// TIA Portal V17 export
// export: Created 2025-03-07T09:18:54.2886173Z, ExportSetting WithDefaults, DisplayName Totally Integrated Automation Portal, DisplayVersion V17 Update 8, DisplayName TIA Portal Openness, DisplayVersion V17 Update 8, DisplayName TIA Portal Version Control Interface, DisplayVersion V17, DisplayName SINAMICS Startdrive Advanced, DisplayVersion V17 SP2, DisplayName SINAMICS Startdrive G110M, G120, G120C, G120D, G120P, G115D, DisplayVersion V17 SP2, DisplayName SINAMICS Startdrive G130, G150, S120, S150, SINAMICS MV, S210, DisplayVersion V17 SP2, DisplayName STEP 7 Professional, DisplayVersion V17 Update 8, DisplayName SINUMERIK ONE STEP 7 Toolbox, DisplayVersion V17 Update 12, DisplayName SINUMERIK 840D sl STEP 7 Toolbox, DisplayVersion V17 Update 12, DisplayName STEP 7 Safety, DisplayVersion V17 Update 6, DisplayName WinCC Advanced, DisplayVersion V17 Update 8
DATA_BLOCK "DB20211_TRUMPF_LASER_UNIT_02_READY"   // DB20211
{ DB_Accessible_From_OPC_UA := 'FALSE' }
VERSION : 0.1
// stored: AutoNumber false, DBAccessibleFromOPCUA false, DBAccessibleFromWebserver true, InstanceOfName FB20200_TRUMPF_READY, InstanceOfType FB
"FB20200_TRUMPF_READY"
   // VAR_INPUT
   //    iLIMIT_MIN_POWER : Int;
   //    iLIMIT_MAX_POWER : Int;
   //    iCOMMAND_POWER : Int;
   //    iCOMMAND_PROCESSING : Int;
   //    iCOMMAND_POWER_PORTION_CORE : Int;
   //    iSTATUS_READY_LASER_READY : Bool;
   //    iLASER_IS_ON : Bool;
   //    iSYSTEM_ERROR_LASER_FAULT : Bool;
   //    iEXTERNAL_CONTROL_READY : Bool;
   //    iPROGRAM_ACTIVE : Bool;
   //    iSOURCE_ENABLED : Bool;
   //    iCOOLING_UNIT_FLOW_PRESENT : Bool;
   //    iCOOLING_UNIT_OVERTEMPERATURE : Bool;
   //    iLASER_ENABLE_POWER_SEQ : Bool;
   //    iLASER_DISABLE_POWER_SEQ : Bool;
   //    iSAFETY_GATES_CLOSED_LOCKED : Bool;
   //    iLASER_ASSIGNED : Bool;
   //    iMACHINE_ON : Bool;
   //    iMACHINE_ON_DELAYED : Bool;
   //    iLASER_READY_F_CIRCUIT_BRAKER : Bool;
   //    iLASER_WARNING_LAP_ON : Bool;
   //    iSTATION_UNIT_ANY_CYCLE_ACT : Bool;
   //    iLASER_ACT_START_GEN_CONDITION : Bool;
   //    iUNIT_NO : Byte;
   // END_VAR
   // VAR_OUTPUT
   //    oLIGHT_PATH : Byte;
   //    oPROGRAM_NUMBER : Byte;
   //    oPOWER_VALUE : DInt;
   //    oPROCESSING_VALUE : DInt;
   //    oPOWER_PORTION_CORE_VALUE : DInt;
   //    oLASER_RESET_FAULT_ERROR : Bool;
   //    oLASER_REQUEST : Bool;
   //    oEXTERNAL_CONTROL : Bool;
   //    oLASER_ON : Bool;
   //    oLASER_ARM : Bool;
   //    oSTATION_RHP_SEOC_ALARMS : Bool;
   //    oSTATION_WARNING : Bool;
   //    oREADY_TO_EMISSION : Bool;
   //    oALARM_CIRCUIT_BREAKER_ALARM : Bool;
   //    oALARM_LASER_ERROR : Bool;
   //    oALARM_WARNING_LASER : Bool;
   //    oALARM_LASER_NOT_READY : Bool;
   //    oALARM_LASER_NOT_SWITCHED_ON : Bool;
   //    oALARM_ANALOG_CONTROL_ERROR : Bool;
   //    oALARM_LASER_NOT_ASSIGNED : Bool;
   //    oALARM_OVERTEMPERATURE_ALARM : Bool;
   //    oALARM_LASER_EMERGENCY_STOP_ACTIVE : Bool;
   //    oALARM_LASER_SC_STATUS_ACTIVE : Bool;
   //    oALARM_ACTIVE_PANEL_ERROR : Bool;
   //    oALARM_LASER_MODULE_1_IN_TEST_MODE : Bool;
   //    oALARM_FAULT : Bool;
   // END_VAR
   // VAR RETAIN
   //    DATA { S7_SetPoint := 'True'} : "LASER READY";
   //    "EXT PULSE START REQ" { S7_SetPoint := 'True'} : TON_TIME;
   //    "COOLING UNIT FLOW IN" : Bool;
   //    "COOLING OVERTEMPERATURE IN" : Bool;
   //    "COOLING UNIT FLOW ALARM" : Bool;
   //    "COOLING OVERTEMPERATURE ALARM" : Bool;
   //    INT_AUX : Int;
   // END_VAR
BEGIN
END_DATA_BLOCK
